# EPICS autosave request: acsMotionApp/Db/SPiiPlusMaxParamsRbv_settings.req
$(P)$(M):maxVelocity_RBV.PREC
$(P)$(M):maxAcceleration_RBV.PREC
